ABB RobotStudio station: Solution13.rsstn

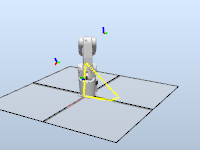
Station Solution13 (saved by RobotStudio 21.4.9700.0)
Controller IRB1200_5_90
  mechanical unit ROB_1: IRB1200_5_90_STD_03_3, 6 joints, base frame (0, 0, 0) mm
Layout (positions relative to the parent item):
  - IRB1200_5_90_STD_03_3 [mechanism, from Robots\IRB1200_5_90_STD_03.rslib] at (0, 0, 0) mm; joint values [0.6076, 0.3838, 1.0157, 0.6147, -1.4304, 3.043] (rad or m)
Targets, tools, work objects and paths stored in the station, written as RAPID:
! task T_ROB1
MODULE Module1
  CONST robtarget Target_10:=[[679.773840836,0,671.640646812],[0.955873065,0,0.293779993,0],[0,0,0,1],[9E+09,9E+09,9E+09,9E+09,9E+09,9E+09]];
  CONST robtarget Target_20:=[[395.070274824,490.545813509,1028.233065681],[0.898252312,0.039361501,-0.082240121,0.429918619],[0,0,-1,1],[9E+09,9E+09,9E+09,9E+09,9E+09,9E+09]];
  CONST jointtarget JointTarget_1:=[[37.05,-7.68,50.04,48.24,-53.86,146.55],[9E+09,9E+09,9E+09,9E+09,9E+09,9E+09]];
  CONST jointtarget JointTarget_2:=[[36.93,-6.61,50.73,47.2,-54.98,148.21],[9E+09,9E+09,9E+09,9E+09,9E+09,9E+09]];
  CONST jointtarget JointTarget_3:=[[36.82,-5.49,51.39,46.19,-56.14,149.85],[9E+09,9E+09,9E+09,9E+09,9E+09,9E+09]];
  CONST jointtarget JointTarget_4:=[[36.71,-4.32,52.03,45.23,-57.35,151.47],[9E+09,9E+09,9E+09,9E+09,9E+09,9E+09]];
  CONST jointtarget JointTarget_5:=[[36.59,-3.09,52.64,44.3,-58.61,153.06],[9E+09,9E+09,9E+09,9E+09,9E+09,9E+09]];
  CONST jointtarget JointTarget_6:=[[36.48,-1.81,53.23,43.41,-59.91,154.63],[9E+09,9E+09,9E+09,9E+09,9E+09,9E+09]];
  CONST jointtarget JointTarget_7:=[[36.37,-0.47,53.79,42.56,-61.25,156.17],[9E+09,9E+09,9E+09,9E+09,9E+09,9E+09]];
  CONST jointtarget JointTarget_8:=[[36.25,0.93,54.32,41.75,-62.63,157.69],[9E+09,9E+09,9E+09,9E+09,9E+09,9E+09]];
  CONST jointtarget JointTarget_9:=[[36.14,2.37,54.82,40.98,-64.05,159.19],[9E+09,9E+09,9E+09,9E+09,9E+09,9E+09]];
  CONST jointtarget JointTarget_11:=[[35.91,5.43,55.74,39.57,-67.01,162.11],[9E+09,9E+09,9E+09,9E+09,9E+09,9E+09]];
  CONST jointtarget JointTarget_12:=[[35.79,7.04,56.15,38.93,-68.54,163.53],[9E+09,9E+09,9E+09,9E+09,9E+09,9E+09]];
  CONST jointtarget JointTarget_13:=[[35.67,8.69,56.53,38.33,-70.09,164.93],[9E+09,9E+09,9E+09,9E+09,9E+09,9E+09]];
  CONST jointtarget JointTarget_14:=[[35.56,10.4,56.87,37.78,-71.68,166.31],[9E+09,9E+09,9E+09,9E+09,9E+09,9E+09]];
  CONST jointtarget JointTarget_15:=[[35.44,12.14,57.18,37.26,-73.28,167.65],[9E+09,9E+09,9E+09,9E+09,9E+09,9E+09]];
  CONST jointtarget JointTarget_16:=[[35.32,13.93,57.45,36.79,-74.9,168.98],[9E+09,9E+09,9E+09,9E+09,9E+09,9E+09]];
  CONST jointtarget JointTarget_17:=[[35.21,15.75,57.69,36.36,-76.54,170.27],[9E+09,9E+09,9E+09,9E+09,9E+09,9E+09]];
  CONST jointtarget JointTarget_18:=[[35.09,17.61,57.89,35.97,-78.18,171.54],[9E+09,9E+09,9E+09,9E+09,9E+09,9E+09]];
  CONST jointtarget JointTarget_19:=[[34.97,19.5,58.05,35.61,-79.82,172.79],[9E+09,9E+09,9E+09,9E+09,9E+09,9E+09]];
  CONST jointtarget JointTarget_21:=[[34.73,23.35,58.25,35.02,-83.11,175.19],[9E+09,9E+09,9E+09,9E+09,9E+09,9E+09]];
  CONST jointtarget JointTarget_22:=[[34.61,25.3,58.3,34.78,-84.74,176.36],[9E+09,9E+09,9E+09,9E+09,9E+09,9E+09]];
  CONST jointtarget JointTarget_23:=[[34.49,27.27,58.3,34.57,-86.35,177.49],[9E+09,9E+09,9E+09,9E+09,9E+09,9E+09]];
  CONST jointtarget JointTarget_24:=[[34.37,29.24,58.27,34.4,-87.94,178.59],[9E+09,9E+09,9E+09,9E+09,9E+09,9E+09]];
  CONST jointtarget JointTarget_25:=[[34.25,31.21,58.2,34.26,-89.51,179.67],[9E+09,9E+09,9E+09,9E+09,9E+09,9E+09]];
  CONST jointtarget JointTarget_26:=[[34.13,33.18,58.09,34.14,-91.05,180.71],[9E+09,9E+09,9E+09,9E+09,9E+09,9E+09]];
  CONST jointtarget JointTarget_27:=[[34.01,35.15,57.93,34.05,-92.56,181.73],[9E+09,9E+09,9E+09,9E+09,9E+09,9E+09]];
  CONST jointtarget JointTarget_28:=[[33.89,37.11,57.75,33.99,-94.03,182.71],[9E+09,9E+09,9E+09,9E+09,9E+09,9E+09]];
  CONST jointtarget JointTarget_29:=[[33.77,39.05,57.52,33.94,-95.46,183.66],[9E+09,9E+09,9E+09,9E+09,9E+09,9E+09]];
  CONST jointtarget JointTarget_30:=[[33.65,40.97,57.26,33.92,-96.84,184.58],[9E+09,9E+09,9E+09,9E+09,9E+09,9E+09]];
  CONST jointtarget JointTarget_31:=[[33.52,42.88,56.96,33.92,-98.19,185.47],[9E+09,9E+09,9E+09,9E+09,9E+09,9E+09]];
  CONST jointtarget JointTarget_32:=[[33.4,44.76,56.62,33.93,-99.48,186.32],[9E+09,9E+09,9E+09,9E+09,9E+09,9E+09]];
  CONST jointtarget JointTarget_33:=[[33.28,46.62,56.26,33.95,-100.73,187.15],[9E+09,9E+09,9E+09,9E+09,9E+09,9E+09]];
  CONST jointtarget JointTarget_34:=[[33.16,48.45,55.85,33.99,-101.93,187.94],[9E+09,9E+09,9E+09,9E+09,9E+09,9E+09]];
  CONST jointtarget JointTarget_35:=[[33.03,50.25,55.42,34.03,-103.08,188.69],[9E+09,9E+09,9E+09,9E+09,9E+09,9E+09]];
  CONST jointtarget JointTarget_36:=[[32.91,52.02,54.95,34.08,-104.18,189.41],[9E+09,9E+09,9E+09,9E+09,9E+09,9E+09]];
  CONST jointtarget JointTarget_37:=[[32.78,53.76,54.46,34.14,-105.23,190.1],[9E+09,9E+09,9E+09,9E+09,9E+09,9E+09]];
  CONST jointtarget JointTarget_38:=[[32.66,55.46,53.93,34.2,-106.24,190.76],[9E+09,9E+09,9E+09,9E+09,9E+09,9E+09]];
  CONST jointtarget JointTarget_39:=[[32.53,57.14,53.38,34.26,-107.19,191.38],[9E+09,9E+09,9E+09,9E+09,9E+09,9E+09]];
  CONST jointtarget JointTarget_40:=[[32.41,58.78,52.8,34.32,-108.09,191.97],[9E+09,9E+09,9E+09,9E+09,9E+09,9E+09]];
  CONST jointtarget JointTarget_41:=[[32.28,60.39,52.2,34.38,-108.95,192.52],[9E+09,9E+09,9E+09,9E+09,9E+09,9E+09]];
  CONST jointtarget JointTarget_42:=[[32.16,61.96,51.56,34.44,-109.75,193.05],[9E+09,9E+09,9E+09,9E+09,9E+09,9E+09]];
  CONST jointtarget JointTarget_43:=[[32.03,63.51,50.91,34.49,-110.52,193.54],[9E+09,9E+09,9E+09,9E+09,9E+09,9E+09]];
  CONST jointtarget JointTarget_44:=[[31.9,65.02,50.23,34.54,-111.24,194],[9E+09,9E+09,9E+09,9E+09,9E+09,9E+09]];
  CONST jointtarget JointTarget_45:=[[31.78,66.51,49.53,34.58,-111.91,194.43],[9E+09,9E+09,9E+09,9E+09,9E+09,9E+09]];
  CONST jointtarget JointTarget_46:=[[31.65,67.96,48.81,34.62,-112.55,194.83],[9E+09,9E+09,9E+09,9E+09,9E+09,9E+09]];
  CONST jointtarget JointTarget_47:=[[31.52,69.38,48.07,34.65,-113.14,195.19],[9E+09,9E+09,9E+09,9E+09,9E+09,9E+09]];
  CONST jointtarget JointTarget_48:=[[31.39,70.78,47.3,34.67,-113.69,195.53],[9E+09,9E+09,9E+09,9E+09,9E+09,9E+09]];
  CONST jointtarget JointTarget_49:=[[31.26,72.15,46.52,34.68,-114.21,195.84],[9E+09,9E+09,9E+09,9E+09,9E+09,9E+09]];
  CONST jointtarget JointTarget_50:=[[32.85,71.82,46.09,36.15,-113.16,196.03],[9E+09,9E+09,9E+09,9E+09,9E+09,9E+09]];
  CONST jointtarget JointTarget_51:=[[34.38,71.48,45.65,37.56,-112.1,196.14],[9E+09,9E+09,9E+09,9E+09,9E+09,9E+09]];
  CONST jointtarget JointTarget_52:=[[35.86,71.14,45.18,38.89,-111.06,196.16],[9E+09,9E+09,9E+09,9E+09,9E+09,9E+09]];
  CONST jointtarget JointTarget_53:=[[37.29,70.8,44.69,40.15,-110.02,196.11],[9E+09,9E+09,9E+09,9E+09,9E+09,9E+09]];
  CONST jointtarget JointTarget_54:=[[38.66,70.47,44.18,41.36,-109,195.99],[9E+09,9E+09,9E+09,9E+09,9E+09,9E+09]];
  CONST jointtarget JointTarget_55:=[[39.99,70.14,43.65,42.51,-108,195.81],[9E+09,9E+09,9E+09,9E+09,9E+09,9E+09]];
  CONST jointtarget JointTarget_56:=[[41.26,69.81,43.1,43.61,-107.01,195.57],[9E+09,9E+09,9E+09,9E+09,9E+09,9E+09]];
  CONST jointtarget JointTarget_57:=[[42.49,69.49,42.53,44.66,-106.05,195.28],[9E+09,9E+09,9E+09,9E+09,9E+09,9E+09]];
  CONST jointtarget JointTarget_58:=[[43.67,69.18,41.94,45.66,-105.11,194.94],[9E+09,9E+09,9E+09,9E+09,9E+09,9E+09]];
  CONST jointtarget JointTarget_59:=[[44.81,68.88,41.33,46.63,-104.19,194.55],[9E+09,9E+09,9E+09,9E+09,9E+09,9E+09]];
  CONST jointtarget JointTarget_60:=[[45.9,68.59,40.71,47.55,-103.3,194.12],[9E+09,9E+09,9E+09,9E+09,9E+09,9E+09]];
  CONST jointtarget JointTarget_61:=[[46.95,68.31,40.07,48.44,-102.43,193.65],[9E+09,9E+09,9E+09,9E+09,9E+09,9E+09]];
  CONST jointtarget JointTarget_62:=[[47.96,68.04,39.41,49.3,-101.59,193.14],[9E+09,9E+09,9E+09,9E+09,9E+09,9E+09]];
  CONST jointtarget JointTarget_63:=[[48.93,67.79,38.74,50.13,-100.77,192.61],[9E+09,9E+09,9E+09,9E+09,9E+09,9E+09]];
  CONST jointtarget JointTarget_64:=[[49.87,67.55,38.05,50.93,-99.98,192.05],[9E+09,9E+09,9E+09,9E+09,9E+09,9E+09]];
  CONST jointtarget JointTarget_65:=[[50.77,67.32,37.34,51.7,-99.21,191.45],[9E+09,9E+09,9E+09,9E+09,9E+09,9E+09]];
  CONST jointtarget JointTarget_66:=[[51.64,67.11,36.62,52.45,-98.47,190.84],[9E+09,9E+09,9E+09,9E+09,9E+09,9E+09]];
  CONST jointtarget JointTarget_67:=[[52.48,66.91,35.88,53.17,-97.75,190.2],[9E+09,9E+09,9E+09,9E+09,9E+09,9E+09]];
  CONST jointtarget JointTarget_68:=[[53.28,66.72,35.13,53.87,-97.05,189.55],[9E+09,9E+09,9E+09,9E+09,9E+09,9E+09]];
  CONST jointtarget JointTarget_69:=[[54.06,66.55,34.36,54.56,-96.38,188.87],[9E+09,9E+09,9E+09,9E+09,9E+09,9E+09]];
  CONST jointtarget JointTarget_70:=[[54.81,66.39,33.58,55.22,-95.73,188.18],[9E+09,9E+09,9E+09,9E+09,9E+09,9E+09]];
  CONST jointtarget JointTarget_71:=[[55.53,66.25,32.79,55.86,-95.1,187.47],[9E+09,9E+09,9E+09,9E+09,9E+09,9E+09]];
  CONST jointtarget JointTarget_72:=[[56.23,66.13,31.98,56.49,-94.5,186.75],[9E+09,9E+09,9E+09,9E+09,9E+09,9E+09]];
  CONST jointtarget JointTarget_73:=[[56.9,66.02,31.16,57.1,-93.91,186.02],[9E+09,9E+09,9E+09,9E+09,9E+09,9E+09]];
  CONST jointtarget JointTarget_74:=[[57.55,65.92,30.32,57.7,-93.35,185.28],[9E+09,9E+09,9E+09,9E+09,9E+09,9E+09]];
  CONST jointtarget JointTarget_75:=[[58.17,65.85,29.47,58.28,-92.8,184.52],[9E+09,9E+09,9E+09,9E+09,9E+09,9E+09]];
  CONST jointtarget JointTarget_76:=[[58.78,65.78,28.61,58.85,-92.28,183.76],[9E+09,9E+09,9E+09,9E+09,9E+09,9E+09]];
  CONST jointtarget JointTarget_77:=[[59.36,65.73,27.74,59.41,-91.77,182.99],[9E+09,9E+09,9E+09,9E+09,9E+09,9E+09]];
  CONST jointtarget JointTarget_78:=[[59.93,65.7,26.85,59.95,-91.28,182.21],[9E+09,9E+09,9E+09,9E+09,9E+09,9E+09]];
  CONST jointtarget JointTarget_79:=[[60.47,65.68,25.95,60.48,-90.8,181.42],[9E+09,9E+09,9E+09,9E+09,9E+09,9E+09]];
  CONST jointtarget JointTarget_80:=[[61,65.68,25.04,61,-90.35,180.62],[9E+09,9E+09,9E+09,9E+09,9E+09,9E+09]];
  CONST jointtarget JointTarget_81:=[[61.51,65.69,24.11,61.51,-89.9,179.82],[9E+09,9E+09,9E+09,9E+09,9E+09,9E+09]];
  CONST jointtarget JointTarget_82:=[[62.01,65.71,23.17,62.01,-89.48,179.02],[9E+09,9E+09,9E+09,9E+09,9E+09,9E+09]];
  CONST jointtarget JointTarget_83:=[[62.49,65.75,22.22,62.5,-89.07,178.2],[9E+09,9E+09,9E+09,9E+09,9E+09,9E+09]];
  CONST jointtarget JointTarget_84:=[[62.95,65.81,21.26,62.98,-88.67,177.39],[9E+09,9E+09,9E+09,9E+09,9E+09,9E+09]];
  CONST jointtarget JointTarget_85:=[[63.4,65.88,20.28,63.46,-88.28,176.57],[9E+09,9E+09,9E+09,9E+09,9E+09,9E+09]];
  CONST jointtarget JointTarget_86:=[[63.84,65.96,19.3,63.92,-87.91,175.74],[9E+09,9E+09,9E+09,9E+09,9E+09,9E+09]];
  CONST jointtarget JointTarget_87:=[[64.26,66.06,18.29,64.37,-87.55,174.91],[9E+09,9E+09,9E+09,9E+09,9E+09,9E+09]];
  CONST jointtarget JointTarget_88:=[[64.68,66.17,17.28,64.82,-87.2,174.07],[9E+09,9E+09,9E+09,9E+09,9E+09,9E+09]];
  CONST jointtarget JointTarget_89:=[[65.07,66.29,16.25,65.26,-86.87,173.24],[9E+09,9E+09,9E+09,9E+09,9E+09,9E+09]];
  CONST jointtarget JointTarget_90:=[[65.46,66.43,15.22,65.69,-86.54,172.39],[9E+09,9E+09,9E+09,9E+09,9E+09,9E+09]];
  CONST jointtarget JointTarget_91:=[[65.84,66.59,14.16,66.12,-86.23,171.55],[9E+09,9E+09,9E+09,9E+09,9E+09,9E+09]];
  CONST jointtarget JointTarget_92:=[[66.2,66.75,13.1,66.53,-85.92,170.7],[9E+09,9E+09,9E+09,9E+09,9E+09,9E+09]];
  CONST jointtarget JointTarget_93:=[[66.56,66.93,12.02,66.95,-85.63,169.84],[9E+09,9E+09,9E+09,9E+09,9E+09,9E+09]];
  CONST jointtarget JointTarget_94:=[[66.9,67.13,10.92,67.35,-85.34,168.98],[9E+09,9E+09,9E+09,9E+09,9E+09,9E+09]];
  CONST jointtarget JointTarget_95:=[[67.24,67.33,9.82,67.75,-85.06,168.12],[9E+09,9E+09,9E+09,9E+09,9E+09,9E+09]];
  CONST jointtarget JointTarget_96:=[[67.57,67.56,8.7,68.15,-84.8,167.26],[9E+09,9E+09,9E+09,9E+09,9E+09,9E+09]];
  CONST jointtarget JointTarget_97:=[[67.88,67.79,7.56,68.54,-84.54,166.39],[9E+09,9E+09,9E+09,9E+09,9E+09,9E+09]];
  CONST jointtarget JointTarget_98:=[[68.19,68.04,6.41,68.92,-84.28,165.51],[9E+09,9E+09,9E+09,9E+09,9E+09,9E+09]];
  CONST jointtarget JointTarget_99:=[[68.49,68.3,5.24,69.3,-84.04,164.63],[9E+09,9E+09,9E+09,9E+09,9E+09,9E+09]];
  CONST jointtarget JointTarget_100:=[[68.73,68.29,5.17,69.53,-84.07,164.53],[9E+09,9E+09,9E+09,9E+09,9E+09,9E+09]];
  CONST jointtarget JointTarget_101:=[[68.97,68.27,5.11,69.77,-84.11,164.43],[9E+09,9E+09,9E+09,9E+09,9E+09,9E+09]];
  CONST jointtarget JointTarget_102:=[[69.2,68.26,5.04,70.01,-84.14,164.33],[9E+09,9E+09,9E+09,9E+09,9E+09,9E+09]];
  CONST jointtarget JointTarget_103:=[[69.44,68.25,4.97,70.25,-84.18,164.23],[9E+09,9E+09,9E+09,9E+09,9E+09,9E+09]];
  CONST jointtarget JointTarget_104:=[[69.67,68.23,4.9,70.48,-84.21,164.13],[9E+09,9E+09,9E+09,9E+09,9E+09,9E+09]];
  CONST jointtarget JointTarget_105:=[[69.91,68.22,4.82,70.72,-84.25,164.02],[9E+09,9E+09,9E+09,9E+09,9E+09,9E+09]];
  CONST jointtarget JointTarget_106:=[[70.15,68.21,4.75,70.95,-84.29,163.92],[9E+09,9E+09,9E+09,9E+09,9E+09,9E+09]];
  CONST jointtarget JointTarget_107:=[[70.38,68.2,4.67,71.19,-84.32,163.81],[9E+09,9E+09,9E+09,9E+09,9E+09,9E+09]];
  CONST jointtarget JointTarget_108:=[[70.61,68.19,4.59,71.42,-84.36,163.7],[9E+09,9E+09,9E+09,9E+09,9E+09,9E+09]];
  CONST jointtarget JointTarget_109:=[[70.85,68.18,4.51,71.66,-84.4,163.6],[9E+09,9E+09,9E+09,9E+09,9E+09,9E+09]];
  CONST jointtarget JointTarget_110:=[[71.08,68.17,4.43,71.89,-84.44,163.49],[9E+09,9E+09,9E+09,9E+09,9E+09,9E+09]];
  CONST jointtarget JointTarget_111:=[[71.31,68.16,4.35,72.12,-84.47,163.38],[9E+09,9E+09,9E+09,9E+09,9E+09,9E+09]];
  CONST jointtarget JointTarget_112:=[[71.54,68.15,4.26,72.35,-84.51,163.27],[9E+09,9E+09,9E+09,9E+09,9E+09,9E+09]];
  CONST jointtarget JointTarget_113:=[[71.78,68.14,4.18,72.58,-84.55,163.16],[9E+09,9E+09,9E+09,9E+09,9E+09,9E+09]];
  CONST jointtarget JointTarget_114:=[[72.01,68.13,4.09,72.81,-84.59,163.04],[9E+09,9E+09,9E+09,9E+09,9E+09,9E+09]];
  CONST jointtarget JointTarget_115:=[[72.24,68.13,4,73.04,-84.63,162.93],[9E+09,9E+09,9E+09,9E+09,9E+09,9E+09]];
  CONST jointtarget JointTarget_116:=[[72.47,68.12,3.91,73.27,-84.67,162.81],[9E+09,9E+09,9E+09,9E+09,9E+09,9E+09]];
  CONST jointtarget JointTarget_117:=[[72.7,68.11,3.82,73.5,-84.71,162.7],[9E+09,9E+09,9E+09,9E+09,9E+09,9E+09]];
  CONST jointtarget JointTarget_118:=[[72.92,68.11,3.72,73.73,-84.75,162.58],[9E+09,9E+09,9E+09,9E+09,9E+09,9E+09]];
  CONST jointtarget JointTarget_119:=[[73.15,68.1,3.63,73.96,-84.79,162.46],[9E+09,9E+09,9E+09,9E+09,9E+09,9E+09]];
  CONST jointtarget JointTarget_120:=[[73.38,68.1,3.53,74.18,-84.83,162.35],[9E+09,9E+09,9E+09,9E+09,9E+09,9E+09]];
  CONST jointtarget JointTarget_121:=[[73.61,68.09,3.43,74.41,-84.87,162.23],[9E+09,9E+09,9E+09,9E+09,9E+09,9E+09]];
  CONST jointtarget JointTarget_122:=[[73.83,68.09,3.33,74.64,-84.91,162.11],[9E+09,9E+09,9E+09,9E+09,9E+09,9E+09]];
  CONST jointtarget JointTarget_123:=[[74.06,68.09,3.22,74.86,-84.95,161.98],[9E+09,9E+09,9E+09,9E+09,9E+09,9E+09]];
  CONST jointtarget JointTarget_124:=[[74.28,68.09,3.12,75.08,-84.99,161.86],[9E+09,9E+09,9E+09,9E+09,9E+09,9E+09]];
  CONST jointtarget JointTarget_125:=[[74.51,68.08,3.01,75.31,-85.04,161.74],[9E+09,9E+09,9E+09,9E+09,9E+09,9E+09]];
  CONST jointtarget JointTarget_126:=[[74.73,68.08,2.91,75.53,-85.08,161.61],[9E+09,9E+09,9E+09,9E+09,9E+09,9E+09]];
  CONST jointtarget JointTarget_127:=[[74.96,68.08,2.8,75.75,-85.12,161.49],[9E+09,9E+09,9E+09,9E+09,9E+09,9E+09]];
  CONST jointtarget JointTarget_128:=[[75.18,68.08,2.69,75.97,-85.17,161.36],[9E+09,9E+09,9E+09,9E+09,9E+09,9E+09]];
  CONST jointtarget JointTarget_129:=[[75.4,68.08,2.58,76.19,-85.21,161.24],[9E+09,9E+09,9E+09,9E+09,9E+09,9E+09]];
  CONST jointtarget JointTarget_130:=[[75.62,68.08,2.46,76.41,-85.26,161.11],[9E+09,9E+09,9E+09,9E+09,9E+09,9E+09]];
  CONST jointtarget JointTarget_131:=[[75.84,68.08,2.35,76.63,-85.3,160.98],[9E+09,9E+09,9E+09,9E+09,9E+09,9E+09]];
  CONST jointtarget JointTarget_132:=[[76.06,68.08,2.23,76.85,-85.35,160.85],[9E+09,9E+09,9E+09,9E+09,9E+09,9E+09]];
  CONST jointtarget JointTarget_133:=[[76.28,68.09,2.11,77.07,-85.39,160.72],[9E+09,9E+09,9E+09,9E+09,9E+09,9E+09]];
  CONST jointtarget JointTarget_134:=[[76.5,68.09,1.99,77.28,-85.44,160.59],[9E+09,9E+09,9E+09,9E+09,9E+09,9E+09]];
  CONST jointtarget JointTarget_135:=[[76.72,68.09,1.87,77.5,-85.49,160.46],[9E+09,9E+09,9E+09,9E+09,9E+09,9E+09]];
  CONST jointtarget JointTarget_136:=[[76.94,68.1,1.74,77.71,-85.53,160.32],[9E+09,9E+09,9E+09,9E+09,9E+09,9E+09]];
  CONST jointtarget JointTarget_137:=[[77.16,68.1,1.62,77.93,-85.58,160.19],[9E+09,9E+09,9E+09,9E+09,9E+09,9E+09]];
  CONST jointtarget JointTarget_138:=[[77.37,68.11,1.49,78.14,-85.63,160.05],[9E+09,9E+09,9E+09,9E+09,9E+09,9E+09]];
  CONST jointtarget JointTarget_139:=[[77.59,68.11,1.36,78.35,-85.68,159.92],[9E+09,9E+09,9E+09,9E+09,9E+09,9E+09]];
  CONST jointtarget JointTarget_140:=[[77.8,68.12,1.23,78.57,-85.73,159.78],[9E+09,9E+09,9E+09,9E+09,9E+09,9E+09]];
  CONST jointtarget JointTarget_141:=[[78.02,68.13,1.1,78.78,-85.78,159.64],[9E+09,9E+09,9E+09,9E+09,9E+09,9E+09]];
  CONST jointtarget JointTarget_142:=[[78.23,68.13,0.97,78.99,-85.83,159.51],[9E+09,9E+09,9E+09,9E+09,9E+09,9E+09]];
  CONST jointtarget JointTarget_143:=[[78.45,68.14,0.83,79.2,-85.88,159.37],[9E+09,9E+09,9E+09,9E+09,9E+09,9E+09]];
  CONST jointtarget JointTarget_144:=[[78.66,68.15,0.7,79.4,-85.93,159.23],[9E+09,9E+09,9E+09,9E+09,9E+09,9E+09]];
  CONST jointtarget JointTarget_145:=[[78.87,68.16,0.56,79.61,-85.98,159.09],[9E+09,9E+09,9E+09,9E+09,9E+09,9E+09]];
  CONST jointtarget JointTarget_146:=[[79.08,68.17,0.42,79.82,-86.04,158.94],[9E+09,9E+09,9E+09,9E+09,9E+09,9E+09]];
  CONST jointtarget JointTarget_147:=[[79.29,68.18,0.28,80.02,-86.09,158.8],[9E+09,9E+09,9E+09,9E+09,9E+09,9E+09]];
  CONST jointtarget JointTarget_148:=[[79.5,68.19,0.14,80.23,-86.14,158.66],[9E+09,9E+09,9E+09,9E+09,9E+09,9E+09]];
  CONST jointtarget JointTarget_149:=[[79.71,68.2,-0.01,80.43,-86.2,158.51],[9E+09,9E+09,9E+09,9E+09,9E+09,9E+09]];
  CONST jointtarget JointTarget_150:=[[79.38,66.87,1.88,80.08,-86.17,159.08],[9E+09,9E+09,9E+09,9E+09,9E+09,9E+09]];
  CONST jointtarget JointTarget_151:=[[79.03,65.54,3.72,79.73,-86.14,159.62],[9E+09,9E+09,9E+09,9E+09,9E+09,9E+09]];
  CONST jointtarget JointTarget_152:=[[78.68,64.22,5.53,79.36,-86.1,160.12],[9E+09,9E+09,9E+09,9E+09,9E+09,9E+09]];
  CONST jointtarget JointTarget_153:=[[78.31,62.9,7.3,78.99,-86.07,160.58],[9E+09,9E+09,9E+09,9E+09,9E+09,9E+09]];
  CONST jointtarget JointTarget_154:=[[77.94,61.58,9.04,78.61,-86.02,161.02],[9E+09,9E+09,9E+09,9E+09,9E+09,9E+09]];
  CONST jointtarget JointTarget_155:=[[77.55,60.26,10.74,78.21,-85.98,161.41],[9E+09,9E+09,9E+09,9E+09,9E+09,9E+09]];
  CONST jointtarget JointTarget_156:=[[77.16,58.93,12.41,77.81,-85.92,161.77],[9E+09,9E+09,9E+09,9E+09,9E+09,9E+09]];
  CONST jointtarget JointTarget_157:=[[76.75,57.6,14.04,77.4,-85.86,162.1],[9E+09,9E+09,9E+09,9E+09,9E+09,9E+09]];
  CONST jointtarget JointTarget_158:=[[76.33,56.27,15.64,76.98,-85.79,162.39],[9E+09,9E+09,9E+09,9E+09,9E+09,9E+09]];
  CONST jointtarget JointTarget_159:=[[75.9,54.93,17.21,76.55,-85.71,162.65],[9E+09,9E+09,9E+09,9E+09,9E+09,9E+09]];
  CONST jointtarget JointTarget_160:=[[75.45,53.58,18.75,76.11,-85.63,162.86],[9E+09,9E+09,9E+09,9E+09,9E+09,9E+09]];
  CONST jointtarget JointTarget_161:=[[74.99,52.22,20.26,75.66,-85.53,163.04],[9E+09,9E+09,9E+09,9E+09,9E+09,9E+09]];
  CONST jointtarget JointTarget_162:=[[74.51,50.85,21.74,75.19,-85.42,163.18],[9E+09,9E+09,9E+09,9E+09,9E+09,9E+09]];
  CONST jointtarget JointTarget_163:=[[74.02,49.47,23.19,74.72,-85.29,163.29],[9E+09,9E+09,9E+09,9E+09,9E+09,9E+09]];
  CONST jointtarget JointTarget_164:=[[73.52,48.08,24.6,74.23,-85.15,163.35],[9E+09,9E+09,9E+09,9E+09,9E+09,9E+09]];
  CONST jointtarget JointTarget_165:=[[73,46.67,25.99,73.73,-85,163.37],[9E+09,9E+09,9E+09,9E+09,9E+09,9E+09]];
  CONST jointtarget JointTarget_166:=[[72.46,45.25,27.34,73.21,-84.82,163.35],[9E+09,9E+09,9E+09,9E+09,9E+09,9E+09]];
  CONST jointtarget JointTarget_167:=[[71.9,43.81,28.66,72.69,-84.63,163.29],[9E+09,9E+09,9E+09,9E+09,9E+09,9E+09]];
  CONST jointtarget JointTarget_168:=[[71.32,42.35,29.95,72.15,-84.41,163.18],[9E+09,9E+09,9E+09,9E+09,9E+09,9E+09]];
  CONST jointtarget JointTarget_169:=[[70.73,40.88,31.21,71.6,-84.17,163.03],[9E+09,9E+09,9E+09,9E+09,9E+09,9E+09]];
  CONST jointtarget JointTarget_170:=[[70.11,39.38,32.43,71.03,-83.9,162.83],[9E+09,9E+09,9E+09,9E+09,9E+09,9E+09]];
  CONST jointtarget JointTarget_171:=[[69.47,37.86,33.62,70.45,-83.61,162.59],[9E+09,9E+09,9E+09,9E+09,9E+09,9E+09]];
  CONST jointtarget JointTarget_172:=[[68.81,36.32,34.78,69.86,-83.28,162.3],[9E+09,9E+09,9E+09,9E+09,9E+09,9E+09]];
  CONST jointtarget JointTarget_173:=[[68.13,34.76,35.9,69.25,-82.91,161.96],[9E+09,9E+09,9E+09,9E+09,9E+09,9E+09]];
  CONST jointtarget JointTarget_174:=[[67.42,33.18,36.98,68.64,-82.51,161.57],[9E+09,9E+09,9E+09,9E+09,9E+09,9E+09]];
  CONST jointtarget JointTarget_175:=[[66.69,31.57,38.02,68.01,-82.07,161.14],[9E+09,9E+09,9E+09,9E+09,9E+09,9E+09]];
  CONST jointtarget JointTarget_176:=[[65.92,29.93,39.03,67.36,-81.58,160.65],[9E+09,9E+09,9E+09,9E+09,9E+09,9E+09]];
  CONST jointtarget JointTarget_177:=[[65.14,28.27,39.99,66.71,-81.04,160.11],[9E+09,9E+09,9E+09,9E+09,9E+09,9E+09]];
  CONST jointtarget JointTarget_178:=[[64.32,26.59,40.91,66.05,-80.45,159.53],[9E+09,9E+09,9E+09,9E+09,9E+09,9E+09]];
  CONST jointtarget JointTarget_179:=[[63.47,24.87,41.79,65.37,-79.81,158.9],[9E+09,9E+09,9E+09,9E+09,9E+09,9E+09]];
  CONST jointtarget JointTarget_180:=[[62.59,23.14,42.62,64.69,-79.11,158.22],[9E+09,9E+09,9E+09,9E+09,9E+09,9E+09]];
  CONST jointtarget JointTarget_181:=[[61.68,21.38,43.41,64,-78.34,157.49],[9E+09,9E+09,9E+09,9E+09,9E+09,9E+09]];
  CONST jointtarget JointTarget_182:=[[60.73,19.6,44.15,63.31,-77.51,156.72],[9E+09,9E+09,9E+09,9E+09,9E+09,9E+09]];
  CONST jointtarget JointTarget_183:=[[59.74,17.79,44.83,62.61,-76.6,155.91],[9E+09,9E+09,9E+09,9E+09,9E+09,9E+09]];
  CONST jointtarget JointTarget_184:=[[58.72,15.97,45.47,61.92,-75.63,155.05],[9E+09,9E+09,9E+09,9E+09,9E+09,9E+09]];
  CONST jointtarget JointTarget_185:=[[57.66,14.14,46.05,61.22,-74.57,154.16],[9E+09,9E+09,9E+09,9E+09,9E+09,9E+09]];
  CONST jointtarget JointTarget_186:=[[56.56,12.29,46.57,60.52,-73.44,153.24],[9E+09,9E+09,9E+09,9E+09,9E+09,9E+09]];
  CONST jointtarget JointTarget_187:=[[55.41,10.43,47.04,59.83,-72.22,152.29],[9E+09,9E+09,9E+09,9E+09,9E+09,9E+09]];
  CONST jointtarget JointTarget_188:=[[54.22,8.56,47.45,59.14,-70.93,151.32],[9E+09,9E+09,9E+09,9E+09,9E+09,9E+09]];
  CONST jointtarget JointTarget_189:=[[52.99,6.7,47.8,58.46,-69.54,150.33],[9E+09,9E+09,9E+09,9E+09,9E+09,9E+09]];
  CONST jointtarget JointTarget_190:=[[51.71,4.85,48.09,57.79,-68.07,149.33],[9E+09,9E+09,9E+09,9E+09,9E+09,9E+09]];
  CONST jointtarget JointTarget_191:=[[50.38,3,48.31,57.13,-66.51,148.33],[9E+09,9E+09,9E+09,9E+09,9E+09,9E+09]];
  CONST jointtarget JointTarget_192:=[[49,1.17,48.47,56.48,-64.86,147.33],[9E+09,9E+09,9E+09,9E+09,9E+09,9E+09]];
  CONST jointtarget JointTarget_193:=[[47.58,-0.63,48.57,55.84,-63.14,146.34],[9E+09,9E+09,9E+09,9E+09,9E+09,9E+09]];
  CONST jointtarget JointTarget_194:=[[46.1,-2.4,48.61,55.21,-61.32,145.36],[9E+09,9E+09,9E+09,9E+09,9E+09,9E+09]];
  CONST jointtarget JointTarget_195:=[[44.57,-4.14,48.58,54.59,-59.43,144.42],[9E+09,9E+09,9E+09,9E+09,9E+09,9E+09]];
  CONST jointtarget JointTarget_196:=[[42.98,-5.83,48.49,53.98,-57.46,143.51],[9E+09,9E+09,9E+09,9E+09,9E+09,9E+09]];
  CONST jointtarget JointTarget_197:=[[41.35,-7.46,48.33,53.37,-55.41,142.64],[9E+09,9E+09,9E+09,9E+09,9E+09,9E+09]];
  CONST jointtarget JointTarget_198:=[[39.66,-9.04,48.11,52.75,-53.3,141.83],[9E+09,9E+09,9E+09,9E+09,9E+09,9E+09]];
  CONST jointtarget JointTarget_199:=[[37.92,-10.56,47.83,52.13,-51.12,141.08],[9E+09,9E+09,9E+09,9E+09,9E+09,9E+09]];
  CONST jointtarget JointTarget_10:=[[36.02,3.88,55.3,40.26,-65.52,160.66],[9E+09,9E+09,9E+09,9E+09,9E+09,9E+09]];
  CONST jointtarget JointTarget_20:=[[34.85,21.42,58.17,35.3,-81.47,174],[9E+09,9E+09,9E+09,9E+09,9E+09,9E+09]];
  CONST jointtarget JointTarget_0:=[[37.16,-8.69,49.34,49.32,-52.79,144.87],[9E+09,9E+09,9E+09,9E+09,9E+09,9E+09]];
  PROC Path_10()
    MoveAbsJ JointTarget_0,v1000,z1,tool0\WObj:=wobj0;
    MoveAbsJ JointTarget_1,v100,z1,tool0\WObj:=wobj0;
    MoveAbsJ JointTarget_2,v100,z1,tool0\WObj:=wobj0;
    MoveAbsJ JointTarget_3,v100,z1,tool0\WObj:=wobj0;
    MoveAbsJ JointTarget_4,v100,z1,tool0\WObj:=wobj0;
    MoveAbsJ JointTarget_5,v100,z1,tool0\WObj:=wobj0;
    MoveAbsJ JointTarget_6,v100,z1,tool0\WObj:=wobj0;
    MoveAbsJ JointTarget_7,v100,z1,tool0\WObj:=wobj0;
    MoveAbsJ JointTarget_8,v100,z1,tool0\WObj:=wobj0;
    MoveAbsJ JointTarget_9,v100,z1,tool0\WObj:=wobj0;
    MoveAbsJ JointTarget_10,v100,z1,tool0\WObj:=wobj0;
    MoveAbsJ JointTarget_11,v100,z1,tool0\WObj:=wobj0;
    MoveAbsJ JointTarget_12,v100,z1,tool0\WObj:=wobj0;
    MoveAbsJ JointTarget_13,v100,z1,tool0\WObj:=wobj0;
    MoveAbsJ JointTarget_14,v100,z1,tool0\WObj:=wobj0;
    MoveAbsJ JointTarget_15,v100,z1,tool0\WObj:=wobj0;
    MoveAbsJ JointTarget_16,v100,z1,tool0\WObj:=wobj0;
    MoveAbsJ JointTarget_17,v100,z1,tool0\WObj:=wobj0;
    MoveAbsJ JointTarget_18,v100,z1,tool0\WObj:=wobj0;
    MoveAbsJ JointTarget_19,v100,z1,tool0\WObj:=wobj0;
    MoveAbsJ JointTarget_20,v100,z1,tool0\WObj:=wobj0;
    MoveAbsJ JointTarget_21,v100,z1,tool0\WObj:=wobj0;
    MoveAbsJ JointTarget_22,v100,z1,tool0\WObj:=wobj0;
    MoveAbsJ JointTarget_23,v100,z1,tool0\WObj:=wobj0;
    MoveAbsJ JointTarget_24,v100,z1,tool0\WObj:=wobj0;
    MoveAbsJ JointTarget_25,v100,z1,tool0\WObj:=wobj0;
    MoveAbsJ JointTarget_26,v100,z1,tool0\WObj:=wobj0;
    MoveAbsJ JointTarget_27,v100,z1,tool0\WObj:=wobj0;
    MoveAbsJ JointTarget_28,v100,z1,tool0\WObj:=wobj0;
    MoveAbsJ JointTarget_29,v100,z1,tool0\WObj:=wobj0;
    MoveAbsJ JointTarget_30,v100,z1,tool0\WObj:=wobj0;
    MoveAbsJ JointTarget_31,v100,z1,tool0\WObj:=wobj0;
    MoveAbsJ JointTarget_32,v100,z1,tool0\WObj:=wobj0;
    MoveAbsJ JointTarget_33,v100,z1,tool0\WObj:=wobj0;
    MoveAbsJ JointTarget_34,v100,z1,tool0\WObj:=wobj0;
    MoveAbsJ JointTarget_35,v100,z1,tool0\WObj:=wobj0;
    MoveAbsJ JointTarget_36,v100,z1,tool0\WObj:=wobj0;
    MoveAbsJ JointTarget_37,v100,z1,tool0\WObj:=wobj0;
    MoveAbsJ JointTarget_38,v100,z1,tool0\WObj:=wobj0;
    MoveAbsJ JointTarget_39,v100,z1,tool0\WObj:=wobj0;
    MoveAbsJ JointTarget_40,v100,z1,tool0\WObj:=wobj0;
    MoveAbsJ JointTarget_41,v100,z1,tool0\WObj:=wobj0;
    MoveAbsJ JointTarget_42,v100,z1,tool0\WObj:=wobj0;
    MoveAbsJ JointTarget_43,v100,z1,tool0\WObj:=wobj0;
    MoveAbsJ JointTarget_44,v100,z1,tool0\WObj:=wobj0;
    MoveAbsJ JointTarget_45,v100,z1,tool0\WObj:=wobj0;
    MoveAbsJ JointTarget_46,v100,z1,tool0\WObj:=wobj0;
    MoveAbsJ JointTarget_47,v100,z1,tool0\WObj:=wobj0;
    MoveAbsJ JointTarget_48,v100,z1,tool0\WObj:=wobj0;
    MoveAbsJ JointTarget_49,v100,z1,tool0\WObj:=wobj0;
    MoveAbsJ JointTarget_50,v100,z1,tool0\WObj:=wobj0;
    MoveAbsJ JointTarget_51,v100,z1,tool0\WObj:=wobj0;
    MoveAbsJ JointTarget_52,v100,z1,tool0\WObj:=wobj0;
    MoveAbsJ JointTarget_53,v100,z1,tool0\WObj:=wobj0;
    MoveAbsJ JointTarget_54,v100,z1,tool0\WObj:=wobj0;
    MoveAbsJ JointTarget_55,v100,z1,tool0\WObj:=wobj0;
    MoveAbsJ JointTarget_56,v100,z1,tool0\WObj:=wobj0;
    MoveAbsJ JointTarget_57,v100,z1,tool0\WObj:=wobj0;
    MoveAbsJ JointTarget_58,v100,z1,tool0\WObj:=wobj0;
    MoveAbsJ JointTarget_59,v100,z1,tool0\WObj:=wobj0;
    MoveAbsJ JointTarget_60,v100,z1,tool0\WObj:=wobj0;
    MoveAbsJ JointTarget_61,v100,z1,tool0\WObj:=wobj0;
    MoveAbsJ JointTarget_62,v100,z1,tool0\WObj:=wobj0;
    MoveAbsJ JointTarget_63,v100,z1,tool0\WObj:=wobj0;
    MoveAbsJ JointTarget_64,v100,z1,tool0\WObj:=wobj0;
    MoveAbsJ JointTarget_65,v100,z1,tool0\WObj:=wobj0;
    MoveAbsJ JointTarget_66,v100,z1,tool0\WObj:=wobj0;
    MoveAbsJ JointTarget_67,v100,z1,tool0\WObj:=wobj0;
    MoveAbsJ JointTarget_68,v100,z1,tool0\WObj:=wobj0;
    MoveAbsJ JointTarget_69,v100,z1,tool0\WObj:=wobj0;
    MoveAbsJ JointTarget_70,v100,z1,tool0\WObj:=wobj0;
    MoveAbsJ JointTarget_71,v100,z1,tool0\WObj:=wobj0;
    MoveAbsJ JointTarget_72,v100,z1,tool0\WObj:=wobj0;
    MoveAbsJ JointTarget_73,v100,z1,tool0\WObj:=wobj0;
    MoveAbsJ JointTarget_74,v100,z1,tool0\WObj:=wobj0;
    MoveAbsJ JointTarget_75,v100,z1,tool0\WObj:=wobj0;
    MoveAbsJ JointTarget_76,v100,z1,tool0\WObj:=wobj0;
    MoveAbsJ JointTarget_77,v100,z1,tool0\WObj:=wobj0;
    MoveAbsJ JointTarget_78,v100,z1,tool0\WObj:=wobj0;
    MoveAbsJ JointTarget_79,v100,z1,tool0\WObj:=wobj0;
    MoveAbsJ JointTarget_80,v100,z1,tool0\WObj:=wobj0;
    MoveAbsJ JointTarget_81,v100,z1,tool0\WObj:=wobj0;
    MoveAbsJ JointTarget_82,v100,z1,tool0\WObj:=wobj0;
    MoveAbsJ JointTarget_83,v100,z1,tool0\WObj:=wobj0;
    MoveAbsJ JointTarget_84,v100,z1,tool0\WObj:=wobj0;
    MoveAbsJ JointTarget_85,v100,z1,tool0\WObj:=wobj0;
    MoveAbsJ JointTarget_86,v100,z1,tool0\WObj:=wobj0;
    MoveAbsJ JointTarget_87,v100,z1,tool0\WObj:=wobj0;
    MoveAbsJ JointTarget_88,v100,z1,tool0\WObj:=wobj0;
    MoveAbsJ JointTarget_89,v100,z1,tool0\WObj:=wobj0;
    MoveAbsJ JointTarget_90,v100,z1,tool0\WObj:=wobj0;
    MoveAbsJ JointTarget_91,v100,z1,tool0\WObj:=wobj0;
    MoveAbsJ JointTarget_92,v100,z1,tool0\WObj:=wobj0;
    MoveAbsJ JointTarget_93,v100,z1,tool0\WObj:=wobj0;
    MoveAbsJ JointTarget_94,v100,z1,tool0\WObj:=wobj0;
    MoveAbsJ JointTarget_95,v100,z1,tool0\WObj:=wobj0;
    MoveAbsJ JointTarget_96,v100,z1,tool0\WObj:=wobj0;
    MoveAbsJ JointTarget_97,v100,z1,tool0\WObj:=wobj0;
    MoveAbsJ JointTarget_98,v100,z1,tool0\WObj:=wobj0;
    MoveAbsJ JointTarget_99,v100,z1,tool0\WObj:=wobj0;
    MoveAbsJ JointTarget_100,v100,z1,tool0\WObj:=wobj0;
    MoveAbsJ JointTarget_101,v100,z1,tool0\WObj:=wobj0;
    MoveAbsJ JointTarget_102,v100,z1,tool0\WObj:=wobj0;
    MoveAbsJ JointTarget_103,v100,z1,tool0\WObj:=wobj0;
    MoveAbsJ JointTarget_104,v100,z1,tool0\WObj:=wobj0;
    MoveAbsJ JointTarget_105,v100,z1,tool0\WObj:=wobj0;
    MoveAbsJ JointTarget_106,v100,z1,tool0\WObj:=wobj0;
    MoveAbsJ JointTarget_107,v100,z1,tool0\WObj:=wobj0;
    MoveAbsJ JointTarget_108,v100,z1,tool0\WObj:=wobj0;
    MoveAbsJ JointTarget_109,v100,z1,tool0\WObj:=wobj0;
    MoveAbsJ JointTarget_110,v100,z1,tool0\WObj:=wobj0;
    MoveAbsJ JointTarget_111,v100,z1,tool0\WObj:=wobj0;
    MoveAbsJ JointTarget_112,v100,z1,tool0\WObj:=wobj0;
    MoveAbsJ JointTarget_113,v100,z1,tool0\WObj:=wobj0;
    MoveAbsJ JointTarget_114,v100,z1,tool0\WObj:=wobj0;
    MoveAbsJ JointTarget_115,v100,z1,tool0\WObj:=wobj0;
    MoveAbsJ JointTarget_116,v100,z1,tool0\WObj:=wobj0;
    MoveAbsJ JointTarget_117,v100,z1,tool0\WObj:=wobj0;
    MoveAbsJ JointTarget_118,v100,z1,tool0\WObj:=wobj0;
    MoveAbsJ JointTarget_119,v100,z1,tool0\WObj:=wobj0;
    MoveAbsJ JointTarget_120,v100,z1,tool0\WObj:=wobj0;
    MoveAbsJ JointTarget_121,v100,z1,tool0\WObj:=wobj0;
    MoveAbsJ JointTarget_122,v100,z1,tool0\WObj:=wobj0;
    MoveAbsJ JointTarget_123,v100,z1,tool0\WObj:=wobj0;
    MoveAbsJ JointTarget_124,v100,z1,tool0\WObj:=wobj0;
    MoveAbsJ JointTarget_125,v100,z1,tool0\WObj:=wobj0;
    MoveAbsJ JointTarget_126,v100,z1,tool0\WObj:=wobj0;
    MoveAbsJ JointTarget_127,v100,z1,tool0\WObj:=wobj0;
    MoveAbsJ JointTarget_128,v100,z1,tool0\WObj:=wobj0;
    MoveAbsJ JointTarget_129,v100,z1,tool0\WObj:=wobj0;
    MoveAbsJ JointTarget_130,v100,z1,tool0\WObj:=wobj0;
    MoveAbsJ JointTarget_131,v100,z1,tool0\WObj:=wobj0;
    MoveAbsJ JointTarget_132,v100,z1,tool0\WObj:=wobj0;
    MoveAbsJ JointTarget_133,v100,z1,tool0\WObj:=wobj0;
    MoveAbsJ JointTarget_134,v100,z1,tool0\WObj:=wobj0;
    MoveAbsJ JointTarget_135,v100,z1,tool0\WObj:=wobj0;
    MoveAbsJ JointTarget_136,v100,z1,tool0\WObj:=wobj0;
    MoveAbsJ JointTarget_137,v100,z1,tool0\WObj:=wobj0;
    MoveAbsJ JointTarget_138,v100,z1,tool0\WObj:=wobj0;
    MoveAbsJ JointTarget_139,v100,z1,tool0\WObj:=wobj0;
    MoveAbsJ JointTarget_140,v100,z1,tool0\WObj:=wobj0;
    MoveAbsJ JointTarget_141,v100,z1,tool0\WObj:=wobj0;
    MoveAbsJ JointTarget_142,v100,z1,tool0\WObj:=wobj0;
    MoveAbsJ JointTarget_143,v100,z1,tool0\WObj:=wobj0;
    MoveAbsJ JointTarget_144,v100,z1,tool0\WObj:=wobj0;
    MoveAbsJ JointTarget_145,v100,z1,tool0\WObj:=wobj0;
    MoveAbsJ JointTarget_146,v100,z1,tool0\WObj:=wobj0;
    MoveAbsJ JointTarget_147,v100,z1,tool0\WObj:=wobj0;
    MoveAbsJ JointTarget_148,v100,z1,tool0\WObj:=wobj0;
    MoveAbsJ JointTarget_149,v100,z1,tool0\WObj:=wobj0;
    MoveAbsJ JointTarget_150,v100,z1,tool0\WObj:=wobj0;
    MoveAbsJ JointTarget_151,v100,z1,tool0\WObj:=wobj0;
    MoveAbsJ JointTarget_152,v100,z1,tool0\WObj:=wobj0;
    MoveAbsJ JointTarget_153,v100,z1,tool0\WObj:=wobj0;
    MoveAbsJ JointTarget_154,v100,z1,tool0\WObj:=wobj0;
    MoveAbsJ JointTarget_155,v100,z1,tool0\WObj:=wobj0;
    MoveAbsJ JointTarget_156,v100,z1,tool0\WObj:=wobj0;
    MoveAbsJ JointTarget_157,v100,z1,tool0\WObj:=wobj0;
    MoveAbsJ JointTarget_158,v100,z1,tool0\WObj:=wobj0;
    MoveAbsJ JointTarget_159,v100,z1,tool0\WObj:=wobj0;
    MoveAbsJ JointTarget_160,v100,z1,tool0\WObj:=wobj0;
    MoveAbsJ JointTarget_161,v100,z1,tool0\WObj:=wobj0;
    MoveAbsJ JointTarget_162,v100,z1,tool0\WObj:=wobj0;
    MoveAbsJ JointTarget_163,v100,z1,tool0\WObj:=wobj0;
    MoveAbsJ JointTarget_164,v100,z1,tool0\WObj:=wobj0;
    MoveAbsJ JointTarget_165,v100,z1,tool0\WObj:=wobj0;
    MoveAbsJ JointTarget_166,v100,z1,tool0\WObj:=wobj0;
    MoveAbsJ JointTarget_167,v100,z1,tool0\WObj:=wobj0;
    MoveAbsJ JointTarget_168,v100,z1,tool0\WObj:=wobj0;
    MoveAbsJ JointTarget_169,v100,z1,tool0\WObj:=wobj0;
    MoveAbsJ JointTarget_170,v100,z1,tool0\WObj:=wobj0;
    MoveAbsJ JointTarget_171,v100,z1,tool0\WObj:=wobj0;
    MoveAbsJ JointTarget_172,v100,z1,tool0\WObj:=wobj0;
    MoveAbsJ JointTarget_173,v100,z1,tool0\WObj:=wobj0;
    MoveAbsJ JointTarget_174,v100,z1,tool0\WObj:=wobj0;
    MoveAbsJ JointTarget_175,v100,z1,tool0\WObj:=wobj0;
    MoveAbsJ JointTarget_176,v100,z1,tool0\WObj:=wobj0;
    MoveAbsJ JointTarget_177,v100,z1,tool0\WObj:=wobj0;
    MoveAbsJ JointTarget_178,v100,z1,tool0\WObj:=wobj0;
    MoveAbsJ JointTarget_179,v100,z1,tool0\WObj:=wobj0;
    MoveAbsJ JointTarget_180,v100,z1,tool0\WObj:=wobj0;
    MoveAbsJ JointTarget_181,v100,z1,tool0\WObj:=wobj0;
    MoveAbsJ JointTarget_182,v100,z1,tool0\WObj:=wobj0;
    MoveAbsJ JointTarget_183,v100,z1,tool0\WObj:=wobj0;
    MoveAbsJ JointTarget_184,v100,z1,tool0\WObj:=wobj0;
    MoveAbsJ JointTarget_185,v100,z1,tool0\WObj:=wobj0;
    MoveAbsJ JointTarget_186,v100,z1,tool0\WObj:=wobj0;
    MoveAbsJ JointTarget_187,v100,z1,tool0\WObj:=wobj0;
    MoveAbsJ JointTarget_188,v100,z1,tool0\WObj:=wobj0;
    MoveAbsJ JointTarget_189,v100,z1,tool0\WObj:=wobj0;
    MoveAbsJ JointTarget_190,v100,z1,tool0\WObj:=wobj0;
    MoveAbsJ JointTarget_191,v100,z1,tool0\WObj:=wobj0;
    MoveAbsJ JointTarget_192,v100,z1,tool0\WObj:=wobj0;
    MoveAbsJ JointTarget_193,v100,z1,tool0\WObj:=wobj0;
    MoveAbsJ JointTarget_194,v100,z1,tool0\WObj:=wobj0;
    MoveAbsJ JointTarget_195,v100,z1,tool0\WObj:=wobj0;
    MoveAbsJ JointTarget_196,v100,z1,tool0\WObj:=wobj0;
    MoveAbsJ JointTarget_197,v100,z1,tool0\WObj:=wobj0;
    MoveAbsJ JointTarget_198,v100,z1,tool0\WObj:=wobj0;
    MoveAbsJ JointTarget_199,v100,z1,tool0\WObj:=wobj0;
  ENDPROC
  PROC main()
    Path_10;
  ENDPROC
ENDMODULE

